// TwinCAT 3 PLC project PlcProjekt
// ProgramVersion: 3.1.4022.1
// libraries:
//   Tc2_Standard, * (Beckhoff Automation GmbH)
//   Tc2_System, * (Beckhoff Automation GmbH)
//   Tc2_Utilities, * (Beckhoff Automation GmbH)
//   Tc3_Module, * (Beckhoff Automation GmbH)
// project tree:
//   GVLs/ AA.TcGVL (not stored), AI.TcGVL (not stored), Blinker.TcGVL (not stored), DA.TcGVL, DI.TcGVL, Plc_AN.TcGVL, Plc_DIO.TcGVL, _PcToPlc.TcGVL (not stored), _PlcToPc.TcGVL (not stored)
//   / PlcTask.TcTTO (not stored)
//   POUs/ MAIN.TcPOU
//   POUs/Privat/ AlleBitSetzen.TcPOU (not stored), BitLesen.TcPOU (not stored), DatenRangieren.TcPOU, IntegerLesen.TcPOU (not stored), IntegerSchreiben.TcPOU, SystemFunktionen.TcPOU (not stored)
// real-time tasks:
//   TASK PlcTask: cycle T#10ms, priority 20, ADS port 350
// motion (NC):
//   TASK NC-Task 1 SAF: cycle T#2ms, priority 4, ADS port 501
//   TASK NC-Task 1 SVB: cycle T#10ms, priority 8, ADS port 511
//   AXIS Axis 1 (id 1)
//     OtherSettings: AllowMotionCmdToSlave=true
//     encoder EncType=4
//       EncPara: MaxCount=#x0000ffff
//         Inc: RefSoftSyncMask=#x0000ffff
//     drive DrvType=24
//       Analog: ScaleFactorActTorque=0.1
//       TimeComp: TaskDelayCycles=1
//     controller CtrType=1
//       CtrPara: PriorControlFactor=1
//         Observer: BandWidth=20
//   AXIS Axis 2 (id 2)
//     OtherSettings: AllowMotionCmdToSlave=true
//     encoder EncType=4
//       EncPara: MaxCount=#x0000ffff
//         Inc: RefSoftSyncMask=#x0000ffff
//     drive DrvType=24
//       Analog: ScaleFactorActTorque=0.1
//       TimeComp: TaskDelayCycles=1
//     controller CtrType=1
//       CtrPara: PriorControlFactor=1
//         Observer: BandWidth=20
//   AXIS Axis 3 (id 3)
//     OtherSettings: AllowMotionCmdToSlave=true
//     encoder EncType=4
//       EncPara: MaxCount=#x0000ffff
//     drive DrvType=23
//       Analog: ScaleFactorActTorque=0.1
//       TimeComp: TaskDelayCycles=1
//     controller CtrType=1
//       CtrPara: PriorControlFactor=1
//         Observer: BandWidth=20
//   AXIS Axis 4 (id 4)
//     OtherSettings: AllowMotionCmdToSlave=true
//     encoder EncType=4
//       EncPara: MaxCount=#x0000ffff
//     drive DrvType=23
//       Analog: ScaleFactorActTorque=0.1
//       TimeComp: TaskDelayCycles=1
//     controller CtrType=1
//       CtrPara: PriorControlFactor=1
//         Observer: BandWidth=20
//   AXIS Axis 5 (id 5)
//     OtherSettings: AllowMotionCmdToSlave=true
//     encoder EncType=19
//       EncPara: MaxCount=#xffffffff
//     drive DrvType=16
//       DrvPara: MaxCount=#xffffffff
//         Analog: ScaleFactorActTorque=0.1
//         TimeComp: TaskDelayCycles=1
//     controller CtrType=1
//       CtrPara: PriorControlFactor=1
//         Observer: BandWidth=20
//   AXIS Axis 6 (id 6)
//     OtherSettings: AllowMotionCmdToSlave=true
//     encoder EncType=19
//       EncPara: MaxCount=#xffffffff
//     drive DrvType=16
//       DrvPara: MaxCount=#xffffffff
//         Analog: ScaleFactorActTorque=0.1
//         TimeComp: TaskDelayCycles=1
//     controller CtrType=1
//       CtrPara: PriorControlFactor=1
//         Observer: BandWidth=20
// I/O:
//   DEVICE Device 1 (EtherCAT), AmsNetId 192.168.200.220.2.1
//     Klemme 1 (EK1200) [EK1200-5000 EtherCAT Netzteil (2A E-Bus)]
//       Klemme 2 (EL3255) [EL3255 5K. Potentiometerauswertung mit Sensorversorgung]
//       Klemme 3 (EL3255) [EL3255 5K. Potentiometerauswertung mit Sensorversorgung]
//       Klemme 4 (EL9011) [EL9011 Endklemme]
// variable links:
//   PlcProjekt/PlcProjekt Instance <-> Device 1 (EtherCAT)/Term 1 (EK1200)/Term 2 (EL3255)
//     PlcTask Inputs/Plc_AN.AI_1_{1..5} <-> AI Standard Channel {1..5}/Value  (5 links)
//     PlcTask Inputs/Plc_DIO.DI_1_{1..5} <-> AI Standard Channel {1..5}/Status  (5 links)
//   PlcProjekt/PlcProjekt Instance <-> Device 1 (EtherCAT)/Term 1 (EK1200)/Term 3 (EL3255)
//     PlcTask Inputs/Plc_AN.AI_2_{1..5} <-> AI Standard Channel {1..5}/Value  (5 links)
//     PlcTask Inputs/Plc_DIO.DI_2_{1..5} <-> AI Standard Channel {1..5}/Status  (5 links)

// ---- GVLs/DA.TcGVL
{attribute 'qualified_only'}
VAR_GLOBAL
END_VAR

// ---- GVLs/DI.TcGVL
{attribute 'qualified_only'}
VAR_GLOBAL	
END_VAR

// ---- GVLs/Plc_AN.TcGVL
{attribute 'qualified_only'}
VAR_GLOBAL		
	AI_1_1 AT %I*: INT;// Value Potentiometer 1-1
	AI_1_2 AT %I*: INT;// Value Potentiometer 1-2	
	AI_1_3 AT %I*: INT;// Value Potentiometer 1-3
	AI_1_4 AT %I*: INT;// Value Potentiometer 1-4
	AI_1_5 AT %I*: INT;// Value Potentiometer 1-5
	
	AI_2_1 AT %I*: INT;// Value Potentiometer 2-1
	AI_2_2 AT %I*: INT;// Value Potentiometer 2-2	
	AI_2_3 AT %I*: INT;// Value Potentiometer 2-3
	AI_2_4 AT %I*: INT;// Value Potentiometer 2-4
	AI_2_5 AT %I*: INT;// Value Potentiometer 2-5
	
	AQ_1 AT %Q*: INT;// Analogausgang AQ 1
END_VAR

// ---- GVLs/Plc_DIO.TcGVL
{attribute 'qualified_only'}
VAR_GLOBAL
	DI_1_1 	AT %I*: BYTE;	// Status Potentiometer 1-1
	DI_1_2 	AT %I*: BYTE;	// Status Potentiometer 1-2
	DI_1_3 	AT %I*: BYTE;	// Status Potentiometer 1-3
	DI_1_4 	AT %I*: BYTE;	// Status Potentiometer 1-4
	DI_1_5 	AT %I*: BYTE;	// Status Potentiometer 1-5
					
	DI_2_1 	AT %I*: BYTE;	// Status Potentiometer 2-1
	DI_2_2 	AT %I*: BYTE;	// Status Potentiometer 2-2
	DI_2_3 	AT %I*: BYTE;	// Status Potentiometer 2-3
	DI_2_4 	AT %I*: BYTE;	// Status Potentiometer 2-4
	DI_2_5 	AT %I*: BYTE;	// Status Potentiometer 2-5
	
	
	DQ_1 AT %QX100.0: BOOL; 		// Digitaler Ausgang 1
END_VAR

// ---- POUs/MAIN.TcPOU
PROGRAM MAIN
VAR
	SystemFunktionen:SystemFunktionen;
END_VAR

DatenRangieren();		// Nicht löschen
SystemFunktionen();		// Nicht löschen

END_PROGRAM

// ---- POUs/Privat/DatenRangieren.TcPOU
PROGRAM DatenRangieren
VAR	
	VersionsText: STRING := 'Simulation Kraftwerkseinsatz V3.0';
	Potentiometer_1_1 : IntegerSchreiben;
	Potentiometer_1_2 : IntegerSchreiben;
	Potentiometer_1_3 : IntegerSchreiben;
	Potentiometer_1_4 : IntegerSchreiben;
	Potentiometer_1_5 : IntegerSchreiben;
	
	Potentiometer_2_1 : IntegerSchreiben;
	Potentiometer_2_2 : IntegerSchreiben;
	Potentiometer_2_3 : IntegerSchreiben;
	Potentiometer_2_4 : IntegerSchreiben;
	Potentiometer_2_5 : IntegerSchreiben;
END_VAR

STRNCPY (ADR( _plcToPc.PlcToPc[96]), ADR( VersionsText), SIZEOF(VersionsText));

_PlcToPc.PlcToPc[0] := Plc_DIO.DI_1_1;
_PlcToPc.PlcToPc[1] := Plc_DIO.DI_1_2;
_PlcToPc.PlcToPc[2] := Plc_DIO.DI_1_3;
_PlcToPc.PlcToPc[3] := Plc_DIO.DI_1_4;
_PlcToPc.PlcToPc[4] := Plc_DIO.DI_1_5;

_PlcToPc.PlcToPc[5] := Plc_DIO.DI_2_1;
_PlcToPc.PlcToPc[6] := Plc_DIO.DI_2_2;
_PlcToPc.PlcToPc[7] := Plc_DIO.DI_2_3;
_PlcToPc.PlcToPc[8] := Plc_DIO.DI_2_4;
_PlcToPc.PlcToPc[9] := Plc_DIO.DI_2_5;



Potentiometer_1_1(Value:= Plc_AN.AI_1_1, LowByte=> _PlcToPc.PlcToPc[32], HighByte=>_PlcToPc.PlcToPc[33]);
Potentiometer_1_1(Value:= Plc_AN.AI_1_2, LowByte=> _PlcToPc.PlcToPc[34], HighByte=>_PlcToPc.PlcToPc[35]);
Potentiometer_1_1(Value:= Plc_AN.AI_1_3, LowByte=> _PlcToPc.PlcToPc[36], HighByte=>_PlcToPc.PlcToPc[37]);
Potentiometer_1_1(Value:= Plc_AN.AI_1_4, LowByte=> _PlcToPc.PlcToPc[38], HighByte=>_PlcToPc.PlcToPc[39]);
Potentiometer_1_1(Value:= Plc_AN.AI_1_5, LowByte=> _PlcToPc.PlcToPc[40], HighByte=>_PlcToPc.PlcToPc[41]);

Potentiometer_2_1(Value:= Plc_AN.AI_2_1, LowByte=> _PlcToPc.PlcToPc[42], HighByte=>_PlcToPc.PlcToPc[43]);
Potentiometer_2_2(Value:= Plc_AN.AI_2_2, LowByte=> _PlcToPc.PlcToPc[44], HighByte=>_PlcToPc.PlcToPc[45]);
Potentiometer_2_3(Value:= Plc_AN.AI_2_3, LowByte=> _PlcToPc.PlcToPc[46], HighByte=>_PlcToPc.PlcToPc[47]);
Potentiometer_2_4(Value:= Plc_AN.AI_2_4, LowByte=> _PlcToPc.PlcToPc[48], HighByte=>_PlcToPc.PlcToPc[49]);
Potentiometer_2_5(Value:= Plc_AN.AI_2_5, LowByte=> _PlcToPc.PlcToPc[50], HighByte=>_PlcToPc.PlcToPc[51]);

END_PROGRAM

// ---- POUs/Privat/IntegerSchreiben.TcPOU
FUNCTION_BLOCK IntegerSchreiben
VAR_INPUT
	Value: INT;
END_VAR
VAR_OUTPUT
	LowByte: BYTE;
	HighByte: BYTE;
END_VAR
VAR	
END_VAR

LowByte := INT_TO_BYTE(Value);
HighByte := INT_TO_BYTE(Value / 256);

END_FUNCTION_BLOCK
